FUNCTION_BLOCK BinaryActuator_MDL_REQ_GEN
  (* Version 1.0, 2005-11-21, Goran Cengic, Chalmers *)
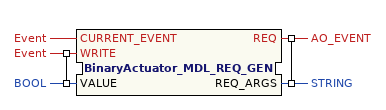
  EVENT_INPUT
    CURRENT_EVENT;
    WRITE WITH VALUE;
  END_EVENT
  EVENT_OUTPUT
    REQ : AO_EVENT WITH REQ_ARGS;
  END_EVENT
  VAR_INPUT
    VALUE : BOOL;
  END_VAR
  VAR_OUTPUT
    REQ_ARGS : STRING;
  END_VAR
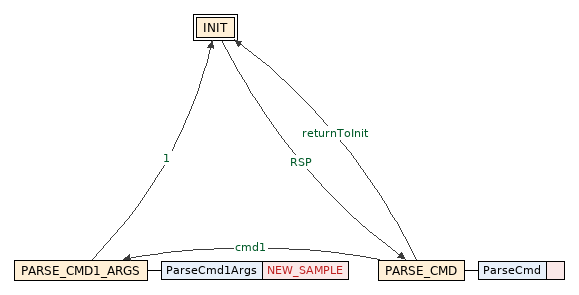
  EC_STATES
    INIT;
    PARSE_CMD : ParseCmd;
    PARSE_CMD1_ARGS : ParseCmd1Args -> NEW_SAMPLE;
  END_STATES
  EC_TRANSITIONS
    INIT TO PARSE_CMD := RSP;
    PARSE_CMD TO PARSE_CMD1_ARGS := cmd1;
    PARSE_CMD TO INIT := returnToInit;
    PARSE_CMD1_ARGS TO INIT := 1;
  END_TRANSITIONS
  ALGORITHM ParseCmd IN Java:
	      cmd = RSP_ARGS.substring(0,RSP_ARGS.indexOf(' '));
	      if (cmd.toLowerCase().equals("new_sample"))
		  {
		    cmd1 = true;
			cmdArgs = RSP_ARGS.substring(RSP_ARGS.indexOf('	') + 1);
		  }
		  else
		  {
		    returnToInit = true;
		  }
  END_ALGORITHM
  ALGORITHM ParseCmd1Args IN Java:
	    NEW_SAMPLE_ARG = (new Boolean(cmdArgs)).booleanValue();
  END_ALGORITHM
END_FUNCTION_BLOCK
